{attribute 'enable_dynamic_creation'}
FUNCTION_BLOCK CMD_LocalMode IMPLEMENTS I_Command
VAR_INPUT
END_VAR
VAR_OUTPUT
END_VAR
VAR
	Comms : I_CommsTransmitter;
	Status : (IDLE, EXECUTE, SENDING, SENT, COMPLETE, TIMED_OUT);
	WatchDog : WatchDog; 
END_VAR
VAR CONSTANT
	CMD : STRING := 'SYSTem:LOCal$R$N';
	TIME_OUT : TIME := T#2S;	
END_VAR

CASE Status OF
	
	EXECUTE: 
		WatchDog.Enable(TIME_OUT);
		Status := SENDING;
		
	SENDING:
		IF Comms.isBusy THEN
			RETURN;
		ELSE
			Comms.Send(CMD);
			Status := SENT;
		END_IF
		
	SENT:
		IF Comms.isBusy THEN
			RETURN;
		ELSE
			WatchDog.Disable();
			Status := COMPLETE;
		END_IF

	IDLE: //
	COMPLETE://
	TIMED_OUT: //
	
END_CASE

IF WatchDog.isTriggered THEN
	WatchDog.Disable();
	Status := TIMED_OUT;
END_IF

METHOD Destroy
VAR_INPUT
END_VAR
VAR
	selfPointer: POINTER TO CMD_LocalMode;
END_VAR
selfPointer := ADR(THIS^);
__DELETE(selfPointer);
END_METHOD

METHOD PUBLIC Execute : BOOL
VAR_INPUT
END_VAR
IF NOT isBusy THEN
	Status := EXECUTE;
	Execute := TRUE;
END_IF

THIS^();
END_METHOD

METHOD FB_init : BOOL
VAR_INPUT
	bInitRetains : BOOL; // if TRUE, the retain variables are initialized (warm start / cold start)
	bInCopyCode : BOOL;  // if TRUE, the instance afterwards gets moved into the copy code (online change)
	Comms : I_CommsTransmitter;
END_VAR
THIS^.Comms := Comms;
END_METHOD

PROPERTY PUBLIC hasTimedOut : BOOL
GET
hasTimedOut := (Status = TIMED_OUT) ;
END_GET
END_PROPERTY

PROPERTY PUBLIC isBusy : BOOL
GET
isBusy := not (Status = IDLE or Status = COMPLETE or Status = TIMED_OUT);
END_GET
END_PROPERTY

PROPERTY isComplete : BOOL
GET
isComplete := (Status = COMPLETE or Status = TIMED_OUT) ;
END_GET
END_PROPERTY

END_FUNCTION_BLOCK

(* stored: Version 1.1.0.1, ProductVersion 3.1.4024.9
   POU CMD_LocalMode: Id {81bd4e41-71f5-4ad9-8da0-df552fed9008}, SpecialFunc None
   Method Destroy: Id {b41c498c-2ecd-4784-a0c6-15ef236441c2}
   Method Execute: Id {ee14a376-4f0b-4d98-aa2e-bf52c5e07060}
   Method FB_init: Id {ea4a2169-70c9-465f-97c6-dc5c4ec9b407}
   Property hasTimedOut: Id {e71f384a-3861-4e27-a9bb-80e9d542a1ff}
   Get Get: Id {953e4562-bbb8-45a1-a7f2-563dbf04758d}
   Property isBusy: Id {4a9a7459-d384-492a-92a8-1c3aae44c0c5}
   Get Get: Id {2eeda75b-c663-4204-9972-29f641f814b1}
   Property isComplete: Id {fc25be20-4579-42c6-9362-a55f518c413f}
   Get Get: Id {7fdd9fca-bcd8-4016-8c6e-34b0a247555d} *)
